FUNCTION_BLOCK CollisionGroup IMPLEMENTS I_Cyclic, I_CollisionGroup, I_Resettable, I_Object
VAR
	stGroupInformation : CAGroupInfo;
	_caGroup : Tc3_McCoordinatedMotion.AXES_GROUP_REF;
	_ICaGroup : I_Mc2CaGroup;
	ReadGroupStatus : Tc3_McCoordinatedMotion.MC_GroupReadStatus;
	ReadErrorCode : Tc3_McCoordinatedMotion.MC_GroupReadError;
	resetCAGroup : ResetGroup := (MyCollisionGroup := THIS^);
	enableCAGroup : EnableGroup := (MyCollisionGroup := THIS^);
	disableCAGroup : DisableGroup := (MyCollisionGroup := THIS^);
	addMover : AddMoverToGroupTask := (MyCollisionGroup := THIS^);
	removeAllAxes : RemoveAllMoverFromGroup := (MyCollisionGroup := THIS^);
	grpStop : StopMoverGroup := (MyCollisionGroup := THIS^);
	removeMover : RemoveMoverFromGroup := (MyCollisionGroup := THIS^);
	_MyName: STRING;
	GroupMovers : ARRAY[0..MaxMovers] OF I_XtsMover;
	RegisteredMovers : INT;
	GroupErrorCode: UDINT;
END_VAR
VAR CONSTANT
	MaxMovers : INT := 49;
END_VAR

{analysis -2}

METHOD AddMoverToThisGroup : HRESULT
VAR_INPUT
	MoverToAdd : I_XtsMover;
END_VAR
VAR
	i : INT;
	Registered : BOOL;
END_VAR
IF MoverToAdd = 0 THEN
	Base_Library.Tracing.Trace.Warning(_MyName, 'Register Mover Fail - null ptr');
	AddMoverToThisGroup := -1;
	RETURN;
END_IF
FOR i := 0 TO MaxMovers DO
	IF GroupMovers[i] = MoverToAdd THEN
		registered := TRUE;
	END_IF
END_FOR
IF registered THEN
	Base_Library.Tracing.Trace.Warning(_MyName, 'Register Mover Fail - registered');
	AddMoverToThisGroup := -2;
	RETURN;
END_IF
IF addMover.Busy THEN
	Base_Library.Tracing.Trace.Warning(_MyName, 'Register Mover Fail - busy');
	AddMoverToThisGroup := -3;
	RETURN;
END_IF

Base_Library.Tracing.Trace.Verbose(_MyName, 'Register Mover Accepted');
addMover.AddMover(MoverToAdd := MoverToAdd);
MoverToAdd.MyCAGroup  := THIS^;
FOR i := 0 TO MaxMovers DO
	IF GroupMovers[i] = 0 THEN
		GroupMovers[i] := MoverToAdd;
		RegisteredMovers := RegisteredMovers + 1;
		EXIT;
	END_IF
END_FOR
END_METHOD

PROPERTY AxisCount : UDINT
GET
AxisCount := _caGroup.NcToPlc.Common.GroupAxesCount;
END_GET
END_PROPERTY

PROPERTY CAGroupXtsIoEnvInterface : I_Mc2CaGroup
GET
CAGroupXtsIoEnvInterface := _ICaGroup;
END_GET
SET
_ICaGroup := CAGroupXtsIoEnvInterface;
IF _ICaGroup <> 0 THEN
	_MyName := _ICaGroup.P_ObjectName;
END_IF
END_SET
END_PROPERTY

METHOD Cycle : HRESULT
VAR
	ResetCaGroupResult : HRESULT;
	EnableCaGroupResult : HRESULT;
	DisableCaGroupResult : HRESULT;
	AddMoverCallResult: HRESULT;
	RemoveAllCycleResult: HRESULT;
	GrpStopCycleResult: HRESULT;
END_VAR
IF _ICaGroup = 0 THEN
	Cycle := -1;
	RETURN;
END_IF


ReadGroupStatus(AxesGroup:= _caGroup, Enable:= TRUE );
ReadErrorCode(AxesGroup := _caGroup, Enable := TRUE, GroupErrorId => GroupErrorCode);
ResetCaGroupResult := resetCAGroup.Cycle();
EnableCaGroupResult := enableCAGroup.Cycle();
DisableCaGroupResult := disableCAGroup.Cycle();
AddMoverCallResult := addMover.Cycle();
RemoveAllCycleResult := removeAllAxes.Cycle();
GrpStopCycleResult := grpStop.Cycle();
removeMover.Cycle();

//Cyclic get CaGroup information
stGroupInformation.sName := 'MainCAGroup';
stGroupInformation.eGroupState := _caGroup.NcToPlc.Common.GroupStatus.State;
stGroupInformation.nAxesCount	:= UDINT_TO_INT(_caGroup.NcToPlc.Common.GroupAxesCount);
stGroupInformation.nId			:= _caGroup.NcToPlc.Common.GroupOID;
END_METHOD

METHOD Disable : BOOL
VAR_INPUT
END_VAR
IF NOT disableCAGroup.Busy THEN
	Base_Library.Tracing.Trace.Verbose(_MyName, 'Group Disable Accepted');
	Disable := SUCCEEDED(disableCAGroup.Execute());
END_IF
END_METHOD

METHOD Enable : BOOL
VAR_INPUT
END_VAR
IF NOT enableCAGroup.Busy THEN
	Base_Library.Tracing.Trace.Verbose(_MyName, 'Group Enable Accepted');
	Enable := SUCCEEDED(enableCAGroup.Execute());
END_IF
END_METHOD

PROPERTY ErrorCode : UDINT
GET
ErrorCode := GroupErrorCode;
END_GET
END_PROPERTY

PROPERTY GroupRef : reference to AXES_GROUP_REF
GET
GroupRef REF= _caGroup;
END_GET
END_PROPERTY

METHOD GroupStop : BOOL
VAR_INPUT
END_VAR
IF NOT grpStop.Busy THEN
	Base_Library.Tracing.Trace.Verbose(_MyName, 'GroupStop accepted');
	GroupStop := SUCCEEDED(grpStop.Execute());
END_IF
END_METHOD

PROPERTY HasError : BOOL
GET
HasError := ReadGroupStatus.GroupErrorStop OR ReadGroupStatus.GroupNotReady;
END_GET
END_PROPERTY

PROPERTY IsDisabled : BOOL
GET
IsDisabled := ReadGroupStatus.GroupDisabled;
END_GET
END_PROPERTY

PROPERTY IsInErrorStop : BOOL
GET
IsInErrorStop := ReadGroupStatus.GroupErrorStop;
END_GET
END_PROPERTY

PROPERTY IsInStandBy : BOOL
GET
IsInStandBy := ReadGroupStatus.GroupStandby;
END_GET
END_PROPERTY

PROPERTY IsMoving : BOOL
GET
IsMoving := ReadGroupStatus.GroupMoving;
END_GET
END_PROPERTY

PROPERTY IsStopping : BOOL
GET
IsStopping := ReadGroupStatus.GroupStopping;
END_GET
END_PROPERTY

PROPERTY MyName : string
GET
MyName := _MyName;
END_GET
END_PROPERTY

METHOD RegisterWithParent
VAR_INPUT
	Parent	: I_HostObjects;
END_VAR
Parent.RegisterCyclic(THIS^);
END_METHOD

METHOD RemoveAllMovers : HRESULT
VAR
	i : INT;
END_VAR
IF removeAllAxes.Busy THEN
	Base_Library.Tracing.Trace.Warning(_MyName, 'Remove All Failed - busy');
	RemoveAllMovers := -1;
	RETURN;
END_IF
IF RegisteredMovers = 0 THEN
	Base_Library.Tracing.Trace.Warning(_MyName, 'Remove All Failed - No Movers');
	RemoveAllMovers := -2;
	RETURN;
END_IF

Base_Library.Tracing.Trace.Verbose(_MyName, 'Remove All Movers Accepted');
removeAllAxes.RemoveAllMover();
RegisteredMovers := 0;
FOR i := 0 TO MaxMovers DO
	GroupMovers[i] := 0;
END_FOR
END_METHOD

METHOD RemoveAMover : HRESULT
VAR_INPUT
	MoverToRemove : I_XtsMover;
END_VAR
VAR
	i : INT;
	registered : BOOL;
END_VAR
IF removeMover.Busy THEN
	Base_Library.Tracing.Trace.Warning(MyName, 'Remove Fail - busy');
	RemoveAMover := -1;
	RETURN;
END_IF
IF MoverToRemove = 0 THEN
	Base_Library.Tracing.Trace.Warning(MyName, 'Remove Fail - null ptr');
	RemoveAMover := -2;
	RETURN;
END_IF
FOR i := 0 TO MaxMovers DO
	IF GroupMovers[i] = MoverToRemove THEN
		registered := TRUE;
	END_IF
END_FOR
IF NOT registered THEN
	Base_Library.Tracing.Trace.Warning(MyName, 'Remove Fail - not registered');
	RemoveAMover := -2;
	RETURN;
END_IF

Base_Library.Tracing.Trace.Verbose(MyName, 'Remove a Mover Accepted');
removeMover.Execute(MoverToRemove.IdentInGroup);
FOR i := 0 TO MaxMovers DO
	IF GroupMovers[i] = MoverToRemove THEN
		GroupMovers[i] := 0;
		RegisteredMovers := RegisteredMovers -1;
	END_IF
END_FOR
END_METHOD

METHOD PUBLIC Reset : HRESULT
IF NOT resetCAGroup.Busy THEN
	Base_Library.Tracing.Trace.Verbose(MyName, 'Group Reset Accepted');
	Reset := resetCAGroup.Execute();
END_IF
END_METHOD

END_FUNCTION_BLOCK

(* stored: Version 1.1.0.1
   POU CollisionGroup: Id {8907fd76-d392-4030-a5c6-041188f5b990}, SpecialFunc None
   Folder Commands: Id {8586cf21-15e1-44d9-a164-c4e3c5e15810}
   Folder Status: Id {f0a1ad0e-7de5-4634-834b-41b20fa92032}
   Method AddMoverToThisGroup: Id {9f418b4e-0cf8-4b65-9d2d-7e6c1a46690c}
   Property AxisCount: Id {b3e2bb0a-a069-4fe7-9ef2-930a2335fa2d}
   Get Get: Id {8a83eac8-ebc4-4ad4-a321-ce4de2a62c2a}
   Property CAGroupXtsIoEnvInterface: Id {212be6c7-141f-4d0f-8757-6216cdee75b6}
   Get Get: Id {58823424-db7c-4e8e-8355-ea0d3f334737}
   Set Set: Id {4e382846-3fb7-428a-a6d3-609bca8b4701}
   Method Cycle: Id {6b3cc58f-cb00-45fb-b855-5eb19dbaab5d}
   Method Disable: Id {236769ac-ee48-442c-86de-25258567af7c}
   Method Enable: Id {9a19e9ba-2611-4357-a3d4-698f998ad87d}
   Property ErrorCode: Id {0223acc2-4094-4ae7-ad44-9e49d1f10cb6}
   Get Get: Id {d01acf5f-5766-4d06-b034-a3a6626d2977}
   Property GroupRef: Id {05d388ea-a899-4954-b35a-8298ecb26dd6}
   Get Get: Id {9960c5ab-7079-4a22-9f43-e4d1a1a5992b}
   Method GroupStop: Id {96e619f0-ba68-4e46-ba5e-bd7a0dcefde6}
   Property HasError: Id {75b1333d-dd26-4f58-89b1-cf0451e8e0c2}
   Get Get: Id {faa780fa-6ea0-4c20-937a-c759ac59f530}
   Property IsDisabled: Id {424ba43e-5002-4522-bd9e-84372637a5ce}
   Get Get: Id {be766286-f53f-468f-9efd-009a74b6d9d7}
   Property IsInErrorStop: Id {797bd075-931c-4132-8262-c07ca523a6de}
   Get Get: Id {fe3739ff-184b-44ae-a8a4-d5835be534ee}
   Property IsInStandBy: Id {d604aabe-599b-4a43-a1c7-efd60e8e3039}
   Get Get: Id {fedab88e-07c1-4230-a4c6-88d93706834c}
   Property IsMoving: Id {b3157892-4e81-4592-a823-fc31ce608269}
   Get Get: Id {63db598a-d2fd-41ae-a9a8-f4b34cc85c3e}
   Property IsStopping: Id {5962f4b9-4447-41f5-bc99-0b620d735be6}
   Get Get: Id {88e53af2-ab20-4dcb-b253-98f15b312093}
   Property MyName: Id {e6811d98-40d4-4440-8374-6ce3386e7963}
   Get Get: Id {e4b2e201-13a7-44e4-888f-38c692b30d08}
   Method RegisterWithParent: Id {0f4efa96-221e-4b5f-b62b-0cd9b26287ac}
   Method RemoveAllMovers: Id {72daaa8f-92d0-4f12-b8f9-45742cf249d6}
   Method RemoveAMover: Id {c380af90-39ac-42df-b7a5-a3aab3a831b8}
   Method Reset: Id {261470fc-03e1-4de0-831a-fe53e2e9126b} *)
